FUNCTION_BLOCK b (* Composite Function Block Type *)
  (* Standard: 61499-2 *)
  (* Version 0.0, 2019-02-09, 4DIAC-IDE, 4DIAC-Consortium *)
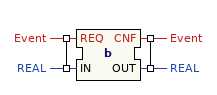
  EVENT_INPUT
    REQ WITH IN; (* Normal Execution Request *)
  END_EVENT
  EVENT_OUTPUT
    CNF WITH OUT; (* Execution Confirmation *)
  END_EVENT
  VAR_INPUT
    IN : REAL;
  END_VAR
  VAR_OUTPUT
    OUT : REAL;
  END_VAR
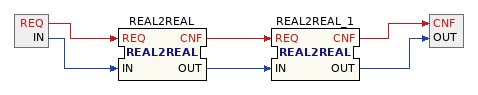
  FBS
    REAL2REAL : REAL2REAL;
    REAL2REAL_1 : REAL2REAL;
  END_FBS
  EVENT_CONNECTIONS
    REAL2REAL.CNF TO REAL2REAL_1.REQ;
    REQ TO REAL2REAL.REQ;
    REAL2REAL_1.CNF TO CNF;
  END_CONNECTIONS
  DATA_CONNECTIONS
    REAL2REAL.OUT TO REAL2REAL_1.IN;
    IN TO REAL2REAL.IN;
    REAL2REAL_1.OUT TO OUT;
  END_CONNECTIONS
END_FUNCTION_BLOCK
